{attribute addProperty Name "AnalogueCheckerData"}
{attribute 'qlik_entity:Checks'}
{attribute 'qlik_ref_value_field:CheckName = AttributeHumanReadable'}
{attribute 'qlik_ref_value_field:StationName = AttributeQlikGroup'}
{attribute 'qlik_value_field:CheckType = Analogue'}
TYPE
    TcoDataInspectorData EXTENDS TcoInspectorData :
    STRUCT
        (*~
		<docu>
		<summary>
			Required status for the check to Pass.	
		</summary>
		</docu>
		~*)
        {attribute addProperty Name "<#Required#>"}
        {attribute 'qlik_load:RequiredStatus'}
        RequiredStatus : STRING(255);

        (*~
		<docu>
		<summary>
			Detected status.	
		</summary>
		</docu>
		~*)
        {attribute addProperty  Name "<#Detected#>"}
        {attribute clr [RenderIgnore("Control", "ShadowControl")]}
        {attribute 'qlik_load:Measured'}
        DetectedStatus : STRING(255);  


		(*~
		<docu>
		<summary>
			When enabled (`true`) the date are evaluating with simple pattern matching.
		</summary>
		</docu>
		~*)
        {attribute addProperty  Name "<*>"}
        {attribute clr [RenderIgnore("Control", "ShadowControl")]}
        {attribute 'qlik_load:Measured'}
		StarNotationEnabled : BOOL;      
    END_STRUCT
END_TYPE

(* stored: Version 1.1.0.1, ProductVersion 3.1.4024.9
   DUT TcoDataInspectorData: Id {07fd2ae7-5bb6-07d4-25b5-19063f05329d} *)
